PROGRAM P_DecAusStossV
VAR
END_VAR

IF DB6.rAusstossverz >= 0.1 THEN
	DB6.rAusstossverz := DB6.rAusstossverz - 0.1;
	DB6.nAusstossverz := REAL_TO_INT(DB6.rAusstossverz * 1000);
END_IF

END_PROGRAM

(* stored: Version 1.1.0.1, ProductVersion 3.1.4024.3
   POU P_DecAusStossV: Id {35672304-a80d-4bd0-a5d5-9096681a96a9}, SpecialFunc None *)
